FUNCTION_BLOCK INTERNAL FB_PathUtilities_Tests EXTENDS FB_TestSuite
VAR_INPUT
END_VAR
VAR_OUTPUT
END_VAR
VAR
	_pathUtilities	: FB_PathUtilities;
END_VAR

Test01_PathExists();
Test02_PathDoesNotExist_ExpectFalseResult();

METHOD Test01_PathExists
VAR_INPUT
END_VAR
VAR
	exists	: BOOL;
END_VAR
IF TcUnit.TEST_ORDERED('Test01_PathExists') THEN
	IF _pathUtilities.Exists(PRG_TESTS.FILE_HANDLER_TESTS_PATH, PRG_TESTS.NET_ID, result => exists) THEN
		AssertTrue(exists, 'Provided path exists, returned result should be TRUE');
		TcUnit.TEST_FINISHED();
	END_IF
END_IF
END_METHOD

METHOD Test02_PathDoesNotExist_ExpectFalseResult
VAR_INPUT
END_VAR
VAR
	exists	: BOOL;
END_VAR
IF TcUnit.TEST_ORDERED('Test02_PathDoesNotExist_ExpectFalseResult') THEN
	IF _pathUtilities.Exists('Some randome path...', '', result => exists) THEN
		AssertFalse(exists, 'Provided path does not exist, returned result should be FALSE.');
		TcUnit.TEST_FINISHED();
	END_IF
END_IF
END_METHOD

END_FUNCTION_BLOCK

(* stored: Version 1.1.0.1, ProductVersion 3.1.4024.15
   POU FB_PathUtilities_Tests: Id {d8d70865-abf7-0ef9-076a-a8b3d2ff3867}, SpecialFunc None
   Method Test01_PathExists: Id {3d495868-8164-04e2-3218-7ecf6076a754}
   Method Test02_PathDoesNotExist_ExpectFalseResult: Id {1bcdcf37-0b53-03cd-1f20-9b3880c594a7} *)
